Staubli VAL3: english.pjx

--- english.pjx ---
Parameters version=s7.1 stackSize=5000 millimeterUnit=true
Program file=message.pgx
Program file=page.pgx
Data file=english.dtx

--- message.pgx ---
public program message(string& message[], num index)
// English PALLET message
begin
  // lenght of message
  //
  switch index
    case 0
      message="change all the approach"
    break
    case 1
      message="change all the depart"
    break
    // NOTE USE MAXIMUN 9 CHAR
    //         012345678
    case 2
      message="Speed"
    break
    case 3
      message="Approach"
    break
    case 4
      message="Depart"
    break
    case 5
      message="App Speed"
    break
    case 6
      message="Dep Speed"
    break
    // NOTE USE MAXIMUN 9 CHAR END
    //         012345678
    case 7
      message="Get at the POINT approach..."
    break
    case 8
      message="Get at the POINT..."
    break
    case 9
      message="Get at the POINT depart..."
    break
    case 10
      message="Get at outside zone point "
    break
    // NOTE USE MAXIMUN 9 CHAR
    //         012345678
    case 11
      message="position "
    break
    case 12
      message="pos.  X  "
    break
    case 13
      message="pos.  Y  "
    break
    case 14
      message="pos.  Z  "
    break
    case 15
      message="on Layer "
    break
    case 16
      message="Select"
    break
    case 17
      message="Press F1 to select the Tool#F8 to continue with the default one: "
    break
    case 18
      message="How many X lines? "
    break
    case 19
      message="How many Y lines? "
    break
    case 20
      message="How many Z lines? "
    break
    case 21
      message="How much is the approach? [mm] "
    break
    case 22
      message="How much is the depart? [mm] "
    break
    case 23
      message="How much is the speed approach? [mm/sec] "
    break
    case 24
      message="How much is the speed depart? [mm/sec] "
    break
    case 25
      message="Do you want a linear move to the point? "
    break
    case 26
      message="Insert the first Instruction,press:#F1 select the instruction#F2 set TCP-> ON #F3 set TCP-> OFF#F8 to END..."
    break
    case 27
      message="Insert the second Instruction,press:#F1 to continue without#F8 to select"
    break
    case 28
      message="How much is the speed? [%]"
    break
    case 29
      message="How much is the speed? [mm/sec]"
    break
    case 30
      message="- Edit to modify the point   "
    break
    case 31
      message="Do you want to validate the last modification ?"
    break
    case 32
      message="Error while computing the frame check your points again"
    break
    //
    case 40
      message="Approach"
    break
    case 41
      message="Depart"
    break
    case 42
      message="tool and point reference (z-)"
    break
    case 43
      message="Stop Time"
    break
  endSwitch
end

--- page.pgx ---
public program page(string& menuname[], num index)
// set all the page in english
begin
  //
  //  PAGE
  //
  //
  // PALLET PAGE
  if index>=10 and index<=19
    title("< Page Pallet >")
  endIf
  // PALLET VIEW PAGE
  if index>=100 and index<=109
    title("< Page View Pallet >")
  endIf
  switch index
    //
    // PALLET
    //
    // Integrator programmer
    case 10,11
      menuname="View Program,Edit Pallet,,,Wizard,Reset,Back,Next"
    break
    // On Cycle
    case 13,14
      menuname="View Program,Edit Pallet,,,,Reset,Back,Next"
    break
    // VIEW PALLET
    case 100,101,102,103,104,105
      menuname="Reset ALL,,,,,Reset,Back,Next"
    break
  endSwitch
end
